// TIA Portal project "encoder" (V14)

(* hardware
DEVICE "HMI_1"  KTP400 Basic PN
   slot 0: "KTP400 Basic PN"  KTP400 Basic PN  6AV2 123-2DB03-0AX0  14.0.1.0
   slot 1: "HMI_RT_1"  KTP400 Basic PN  6AV2 123-2DB03-0AX0  14.0.1.0
   slot 5: "HMI_1.IE_CP_1"  PROFINET Interface  14.0.1.0
      slot 1: "PROFINET Interface_1"  PROFINET Interface
         slot 1: "Port_1"  Port
DEVICE "S7-1200 station_1"  S7-1200 Station
   slot 0: "Rack_0"  S7-1200 Rack  Rack  V1.0
   slot 1: "PLC_1"  CPU 1212C DC/DC/DC  6ES7 212-1AE40-0XB0  V4.2
*)

// ===== PLC "PLC_1"  CPU 1212C DC/DC/DC =====

VAR_GLOBAL   // PLC tag table "Default tag table"
   "Tag_1" AT %M0.2 : Bool;
   "Tag_2" AT %ID1000 : DWord;
   "Tag_3" AT %MD2 : DWord;
   "Tag_4" AT %MD6 : Real;
   "LUULUONG" AT %MD7 : Real;
   "Tag_5" AT %M0.0 : Bool;
   "START" AT %M0.1 : Bool;
   "STOP" AT %M0.3 : Bool;
   "TAM" AT %M0.4 : Bool;
END_VAR

ORGANIZATION_BLOCK "Main"   // OB1, LAD, ProgramCycle
TITLE = "Main Program Sweep (Cycle)"
{ S7_Optimized_Access := 'TRUE' }
VERSION : 0.1
   VAR_INPUT
      Initial_Call : Bool;   // Initial call of this OB
      Remanence : Bool;   // =True, if remanent data are available
   END_VAR
BEGIN

REGION Network 1
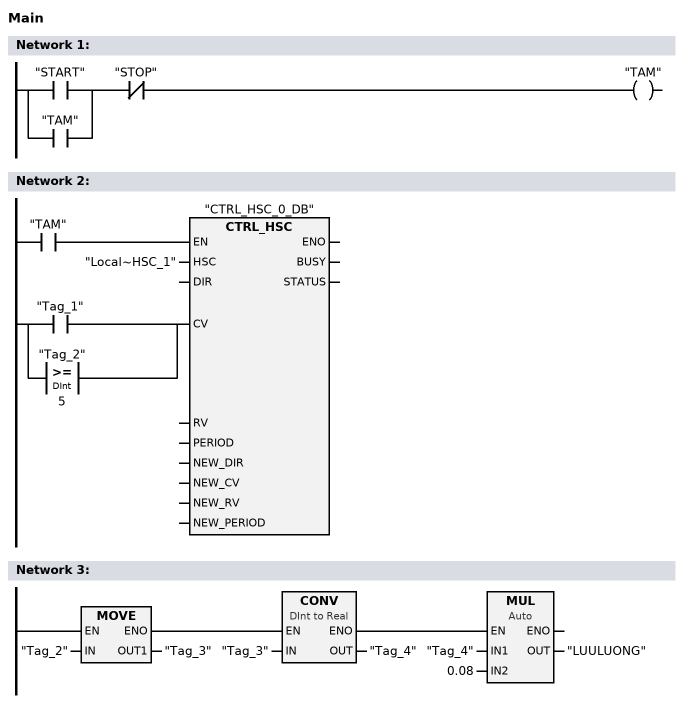
   RUNG wire#powerrail
      Contact( "START" )
      wire#w1
      I_Contact( "STOP" )
      Coil( "TAM" )
   END_RUNG
   RUNG wire#powerrail
      Contact( "TAM" )
   END_RUNG wire#w1
   // the same network as SCL:
   "TAM" := ("START" OR "TAM") AND NOT "STOP";
END_REGION

REGION Network 2
   IF "TAM" THEN
       "CTRL_HSC_0_DB"(HSC := "Local~HSC_1", CV := "Tag_1" OR ("Tag_2" >= 5));   // CTRL_HSC
   END_IF;
END_REGION

REGION Network 3
   RUNG wire#powerrail
      Move(in := "Tag_2", out1 => "Tag_3")
      { S7_Templates := "[SrcType := DInt, DestType := Real]" } Convert(in := "Tag_3", out => "Tag_4")
      Mul(in1 := "Tag_4", in2 := 0.08, out => "LUULUONG")
   END_RUNG
   // the same network as SCL:
   "Tag_3" := "Tag_2";
   "Tag_4" := DINT_TO_REAL("Tag_3");
   "LUULUONG" := "Tag_4" * 0.08;
END_REGION
END_ORGANIZATION_BLOCK

(* ===== HMI "HMI_RT_1" =====
system functions are stored by id; their names below are inferred from use
connection "HMI_Connection_1": ETHERNET, SMART_S7_1200_OMS

HMI tags "Default tag table"
   "TAM" : Bool = PLC TAM AT %M0.4, 1 s
   "START" : Bool = PLC START AT %M0.1, 1 s
   "STOP" : Bool = PLC STOP AT %M0.3, 1 s
   "LUULUONG" : Real = PLC LUULUONG AT %MD7, 1 s

Template "Template_1" 480x272
   Button "Exit" at 388,227 size 63x44; TextOff 'Exit'; PictureOff "ExitRuntime_KTP400_Basic_PN_TR"; PictureOn "ExitRuntime_KTP400_Basic_PN_TR"
      on Release: StopRuntime(0)
   Button "Template_Button" at 268,227 size 63x44; TextOff 'Text'
   Button "Template_Button_1" at 148,227 size 63x44; TextOff 'Text'
   Button "Start screen" at 28,227 size 63x44; TextOff 'Start screen'; PictureOff "NavigateHome_KTP400_Basic_PN_TR"; PictureOn "NavigateHome_KTP400_Basic_PN_TR"
      on Release: ActivateScreen("Root screen", 0)

screen "Root screen" 480x272, template "Template_1"
   TextField "HmiScreenItemData" at 49,9 size 384x22; Text 'DOC LUU LUONG DONG CO MAY BOM'
   Button "Button_1" at 39,102 size 96x32; TextOff 'START'
      on Press: SetBit("START")
      on Release: ResetBit("START")
      Appearance <- "TAM"
   Button "Button_2" at 198,102 size 96x32; TextOff 'STOP'
      on Press: SetBit("STOP")
      on Release: ResetBit("STOP")
      Appearance <- "TAM"
   IOField "I/O field_1" at 318,99 size 96x32; FormatPattern s999999999.999
      ProcessValue <- "LUULUONG"
*)